// TIA Portal V20 export
DATA_BLOCK "LAcycCom_RequestBuffer1"   // DB30500
TITLE = LAcycCom_RequestBuffer
AUTHOR : tech.team.motioncontrol@siemens.com
FAMILY : AcycCom
VERSION : 1.1
// Support: tech.team.motioncontrol@siemens.com
// stored: InstanceOfName LAcycCom_typeRequestBuffer, InstanceOfType UDT, Namespace Unit1.Em2
"LAcycCom_typeRequestBuffer"
   // VAR
   //    header { ExternalWritable := 'False'; S7_SetPoint := 'True'} : "LAcycCom_typeRequestBufferHeader";
   //    elements { ExternalWritable := 'False'; S7_SetPoint := 'True'} : Array[0.."LACYCCOM_BUFFER_ELEMENTS_UPPER_LIM"] of "LAcycCom_typeRequestBufferElement";
   // END_VAR
BEGIN
END_DATA_BLOCK
